FUNCTION_BLOCK "FB_AI"
TITLE = Functional block from AI
{ S7_Optimized_Access := 'FALSE' }
AUTHOR : 'SS&AIs'
FAMILY : Arhive
VERSION : 8.1
// -----------------------------------------------------------------------------
// БЛОК ОБРАБОТКИ АНАЛОГОВОГО СИГНАЛА (FB_AI)
// -----------------------------------------------------------------------------
   VAR_INPUT
      i_iRawSignal { ExternalAccessible := 'False'; ExternalVisible := 'False'; ExternalWritable := 'False'} : Int;
      i_rSimValue { ExternalAccessible := 'False'; ExternalVisible := 'False'; ExternalWritable := 'False'} : Real;
   END_VAR

   VAR_IN_OUT
      io_stConfig : "UDT_AI_Conf";
      io_stOut : "UDT_AI_Out";
   END_VAR

   VAR
      stat_boWasInvalid { ExternalAccessible := 'False'; ExternalVisible := 'False'; ExternalWritable := 'False'} : Bool := TRUE;
   END_VAR

   VAR_TEMP
      temp_rMA : Real;
      temp_rNorm : Real;
      temp_rCutoff_Norm : Real;
      temp_rScaled : Real;
      temp_rRange_mA : Real;
      temp_rRange_Phys : Real;
      temp_rMinPhys : Real;
      temp_rMaxPhys : Real;
      temp_boResetFilter : Bool;
      temp_iFilterTime : Real;
      temp_rHWRange : Real;
      temp_iLimit_Max : Int;
      temp_iLimit_Min : Int;
   END_VAR


BEGIN
	    // =========================================================
	    // ШАГ 0. РАСШИФРОВКА БИТОВОГО СЛОВА (Mode)
	    // =========================================================

	    #io_stOut.Status.Disabled := #io_stConfig.Mode.Disabled;
	    // 0.1 Режим полного отключения канала
	    IF #io_stOut.Status.Disabled THEN
	        #io_stOut.Value_Unclamped := 0.0;
	        #io_stOut.Value_Scaled := 0.0;
	        #io_stOut.Value_Filtered := 0.0;
	        #io_stOut.Value_mA := 0.0;
	        #io_stOut.Raw := 0;

	        #io_stOut.Status.WireBreak := FALSE;
	        #io_stOut.Status.Underrange := FALSE;
	        #io_stOut.Status.Overrange := FALSE;
	        #io_stOut.Status.Overflow := FALSE;
	        #io_stOut.Status.ConfigError := FALSE;
	        #io_stOut.Status.Sim_Active := FALSE;

	        #stat_boWasInvalid := TRUE;
	        RETURN;
	    END_IF;

	    // 0.2 Защита от ошибок конфигурации
	    #temp_rRange_mA := #io_stConfig.Calib_mA_Max - #io_stConfig.Calib_mA_Min;
	    #temp_rRange_Phys := #io_stConfig.Scale_Max - #io_stConfig.Scale_Min;

	    IF (#io_stConfig.HW_Max <= #io_stConfig.HW_Min) OR
	        (#temp_rRange_mA <= 0.0) OR
	        (ABS(#temp_rRange_Phys) < 0.00001) OR
	        (ABS(#io_stConfig.Cutoff) >= ABS(#temp_rRange_Phys)) THEN

	        #io_stOut.Status.ConfigError := TRUE;

	        #io_stOut.Status.WireBreak := FALSE;
	        #io_stOut.Status.Underrange := FALSE;
	        #io_stOut.Status.Overrange := FALSE;
	        #io_stOut.Status.Overflow := FALSE;
	        #io_stOut.Status.Sim_Active := FALSE;

	        #io_stOut.Value_Unclamped := 0.0;
	        #io_stOut.Value_Scaled := 0.0;
	        #io_stOut.Value_Filtered := 0.0;
	        #io_stOut.Value_mA := 0.0;
	        #io_stOut.Raw := #i_iRawSignal;

	        #stat_boWasInvalid := TRUE;
	        RETURN;
	    END_IF;

	    #io_stOut.Status.ConfigError := FALSE;

	    // =========================================================
	    // ШАГ 1 & 2. СИМУЛЯЦИЯ И ДИАГНОСТИКА
	    // =========================================================
	    IF #io_stConfig.Mode.SimActive THEN
	        #io_stOut.Status.Sim_Active := TRUE;

	        #io_stOut.Status.WireBreak := FALSE;
	        #io_stOut.Status.Underrange := FALSE;
	        #io_stOut.Status.Overrange := FALSE;
	        #io_stOut.Status.Overflow := FALSE;

	        #io_stOut.Raw := 0;
	        #io_stOut.Value_mA := 0.0;
	        #temp_rScaled := #i_rSimValue;
	    ELSE
	        #io_stOut.Status.Sim_Active := FALSE;
	        #io_stOut.Raw := #i_iRawSignal;

	        #temp_rHWRange := INT_TO_REAL(#io_stConfig.HW_Max) - INT_TO_REAL(#io_stConfig.HW_Min);

	        //HW диагностика
	        #temp_iLimit_Max := REAL_TO_INT(INT_TO_REAL(#io_stConfig.HW_Min) + ("C_DIAG_OVER" * #temp_rHWRange));
	        #temp_iLimit_Min := REAL_TO_INT(INT_TO_REAL(#io_stConfig.HW_Min) + ("C_DIAG_UNDER" * #temp_rHWRange));

	        #io_stOut.Status.WireBreak := #i_iRawSignal < #temp_iLimit_Min;
	        #io_stOut.Status.Underrange := (#i_iRawSignal < #io_stConfig.HW_Min) AND (#i_iRawSignal >= #temp_iLimit_Min);
	        #io_stOut.Status.Overrange := (#i_iRawSignal > #io_stConfig.HW_Max) AND (#i_iRawSignal <= #temp_iLimit_Max);
	        #io_stOut.Status.Overflow := #i_iRawSignal > #temp_iLimit_Max;

	        // =========================================================
	        // ШАГ 3. МАТЕМАТИКА
	        // =========================================================
	        IF #io_stOut.Status.WireBreak THEN
	            #temp_rScaled := #io_stConfig.Scale_Min + (#temp_rRange_Phys * "C_DIAG_UNDER");
	            #io_stOut.Value_mA := 0.0;

	        ELSIF #io_stOut.Status.Overflow THEN
	            #temp_rScaled := #io_stConfig.Scale_Min + (#temp_rRange_Phys * "C_DIAG_OVER");
	            #io_stOut.Value_mA := 25.0;

	        ELSE
	            // А) Расчет миллиампер
	            #temp_rMA := 4.0 + ((INT_TO_REAL(#i_iRawSignal) - INT_TO_REAL(#io_stConfig.HW_Min)) /
	            #temp_rHWRange) * 16.0;
	            #io_stOut.Value_mA := #temp_rMA;

	            // Б) Нормализация (0.0 ... 1.0)
	            #temp_rNorm := (#temp_rMA - #io_stConfig.Calib_mA_Min) / #temp_rRange_mA;

	            // В & Г) Работа с корнем (Отсечка и извлечение)
	            IF #io_stConfig.Mode.UseSqrt THEN

	                IF #io_stConfig.Mode.PreSqrtCut THEN
	                    #temp_rCutoff_Norm := #io_stConfig.Cutoff / #temp_rRange_Phys;
	                    #temp_rCutoff_Norm := #temp_rCutoff_Norm * #temp_rCutoff_Norm;

	                    IF #temp_rNorm < #temp_rCutoff_Norm THEN
	                        #temp_rNorm := 0.0;
	                    END_IF;
	                END_IF;

	                IF #temp_rNorm > 0.0 THEN
	                    #temp_rNorm := SQRT(#temp_rNorm);
	                ELSE
	                    #temp_rNorm := 0.0;
	                END_IF;

	            END_IF;

	            // Д) Масштабирование в физическую величину
	            #temp_rScaled := #io_stConfig.Scale_Min + (#temp_rNorm * #temp_rRange_Phys);

	            // Е) Классический CutOff (только если не применялся Pre-Sqrt)
	            IF NOT (#io_stConfig.Mode.PreSqrtCut AND #io_stConfig.Mode.UseSqrt) THEN
	                IF ABS(#temp_rScaled) < ABS(#io_stConfig.Cutoff) THEN
	                    #temp_rScaled := 0.0;
	                END_IF;
	            END_IF;
	        END_IF;
	    END_IF;

	    // Сохраняем чистую математику на выход
	    #io_stOut.Value_Unclamped := #temp_rScaled;

	    // =========================================================
	    // ШАГ 3.5. ФИНАЛЬНЫЙ CLAMP
	    // =========================================================
	    IF #io_stConfig.Mode.FinalClamp THEN
	        #temp_rMinPhys := MIN(IN1 := #io_stConfig.Scale_Min, IN2 := #io_stConfig.Scale_Max);
	        #temp_rMaxPhys := MAX(IN1 := #io_stConfig.Scale_Min, IN2 := #io_stConfig.Scale_Max);
	        #temp_rScaled := LIMIT(MN := #temp_rMinPhys, IN := #temp_rScaled, MX := #temp_rMaxPhys);
	    END_IF;

	    #io_stOut.Value_Scaled := #temp_rScaled;

	    // =========================================================
	    // ШАГ 4. ФИЛЬТРАЦИЯ & PRE-LOAD
	    // =========================================================
	    #temp_boResetFilter := #io_stOut.Status.WireBreak OR
	    #io_stOut.Status.Overflow OR
	    #stat_boWasInvalid OR
	    "isFirstScan"();

	    #temp_iFilterTime := INT_TO_REAL(LIMIT(MN := 0, IN := #io_stConfig.FilterTime_ms, MX := 32000));

	    "FC_Filter_PT1"(
	                    i_rRawValue := #temp_rScaled,
	                    i_rTimeFilter_ms := #temp_iFilterTime,
	                    i_boReset := #temp_boResetFilter,
	                    io_rFilteredValue := #io_stOut.Value_Filtered
	    );

	    #stat_boWasInvalid := #io_stOut.Status.WireBreak OR
	    #io_stOut.Status.Overflow OR
	    #io_stOut.Status.ConfigError;

END_FUNCTION_BLOCK

